INTERFACE I_Station EXTENDS I_Resettable, I_Diagnosable

METHOD Execute : BOOL
END_METHOD

PROPERTY State : E_StationState
GET
END_GET
END_PROPERTY

END_INTERFACE

(* stored: Version 1.1.0.1, ProductVersion 3.1.4024.12
   Itf I_Station: Id {0880c320-3eb1-499d-832e-da84b00f8be4}
   Method Execute: Id {f10a79c0-0eb2-4fea-894a-9fc5cb80e5c5}
   Property State: Id {4356f0aa-6568-41b2-85c9-bb82c62f5611}
   Get Get: Id {4edf90df-efca-4ca3-8dc9-f8c0ab2b4f70} *)
